{attribute 'GeneratedUsingTerminal: IODEVICETYPE_ETHERCATPROT'}
{attribute addProperty BoxType "IODEVICETYPE_ETHERCATPROT"}
{attribute addProperty Id "R1_EK1100R1_EK1100_4AD22B7B1143R2_EK1100R2_EK1100_10D8A594458R3_EK1100R3_EK1100_C7887D6C263R4_EK1100R4_EK1100_46A1248C369R4A_EK1100R4A_EK1100_48316913274R5_EK1100R5_EK1100_0007A337146R6_EK1100R6_EK1100_8C41F5F2336R7_EK1100R7_EK1100_F50DDAC8306R8_EK1100R8_EK1100_9C7B3B675648R9_EK1100R9_EK1100_484053C0136R10_EK1100R10_EK1100_C5CE1D87649SyncUnitsSyncUnits_E1A49202432InputsInputs_0514630C40OutputsOutputs_C89C478B26InfoDataInfoData_84133AC922"}
{attribute addProperty CRC "467727330"}
{attribute addProperty Size "10248"}
{attribute addProperty Name "Device 6424 (EtherCAT)"}
TYPE Device_6424_EtherCAT_1BE0F3E2 EXTENDS TcoIo.EtcMasterBase_62654B43 :
STRUCT
	{attribute addProperty Name "R1 (EK1100)"}
	{attribute addProperty PreviousPort "Device 6424 (EtherCAT) : Master"}
	R1_EK1100 : R1_EK1100_4AD22B7B;
	{attribute addProperty Name "R2 (EK1100)"}
	{attribute addProperty PreviousPort "R1 (EK1100) : C"}
	R2_EK1100 : R2_EK1100_10D8A594;
	{attribute addProperty Name "R3 (EK1100)"}
	{attribute addProperty PreviousPort "R2 (EK1100) : C"}
	R3_EK1100 : R3_EK1100_C7887D6C;
	{attribute addProperty Name "R4 (EK1100)"}
	{attribute addProperty PreviousPort "R3 (EK1100) : C"}
	R4_EK1100 : R4_EK1100_46A1248C;
	{attribute addProperty Name "R4A (EK1100)"}
	{attribute addProperty PreviousPort "R4 (EK1100) : C"}
	R4A_EK1100 : R4A_EK1100_48316913;
	{attribute addProperty Name "R5 (EK1100)"}
	{attribute addProperty PreviousPort "R4A (EK1100) : C"}
	R5_EK1100 : R5_EK1100_0007A337;
	{attribute addProperty Name "R6 (EK1100)"}
	{attribute addProperty PreviousPort "R5 (EK1100) : C"}
	R6_EK1100 : R6_EK1100_8C41F5F2;
	{attribute addProperty Name "R7 (EK1100)"}
	{attribute addProperty PreviousPort "R6 (EK1100) : C"}
	R7_EK1100 : R7_EK1100_F50DDAC8;
	{attribute addProperty Name "R8 (EK1100)"}
	{attribute addProperty PreviousPort "R7 (EK1100) : C"}
	R8_EK1100 : R8_EK1100_9C7B3B67;
	{attribute addProperty Name "R9 (EK1100)"}
	{attribute addProperty PreviousPort "R8 (EK1100) : C"}
	R9_EK1100 : R9_EK1100_484053C0;
	{attribute addProperty Name "R10 (EK1100)"}
	{attribute addProperty PreviousPort "R9 (EK1100) : C"}
	R10_EK1100 : R10_EK1100_C5CE1D87;
	{attribute addProperty Name "SyncUnits"}
	SyncUnits : SyncUnits_E1A49202;
	{attribute addProperty Name "Inputs"}
	Inputs : Inputs_0514630C;
	{attribute addProperty Name "Outputs"}
	Outputs : Outputs_C89C478B;
	{attribute addProperty Name "InfoData"}
	InfoData : TcoIo.InfoData_84133AC9;
END_STRUCT
END_TYPE

(* stored: Version 1.2.0.0, ProductVersion 3.1.4024.11
   DUT Device_6424_EtherCAT_1BE0F3E2: Id {4de72bce-b7b2-0dbb-340d-114cc1de9c6a} *)
